TYPE SimpleStepLog :
STRUCT
	number			: LINT;
	name			: STRING;
	description		: T_MaxString;
	duration		: TIME;
	mode			: STRING;
END_STRUCT
END_TYPE

(* stored: Version 1.1.0.1, ProductVersion 3.1.4024.11
   DUT SimpleStepLog: Id {b1d48f56-d758-49eb-b9ac-629105b85570} *)
